(* Logix 5000 project; controller test_calc vendor 1 type 14 code 106 rev 31.11; software revision 31.01 *)

TASK MainTask (continuous, watchdog 500 ms) : MainProgram

MODULES
   Local : vendor 1 type 14 code 106 (Compact 0, rev 31.11)
END_MODULES

VAR_GLOBAL   (* controller tags *)
   cyc_h : REAL;
   cyl_h : REAL;
   cyl_rad : REAL;
   GAL : REAL;
END_VAR

PROGRAM MainProgram   (* main routine MainRoutine *)

ROUTINE calc   (* structured text *)
   pi*cyl_rad^2-cyl_rad^2*ACOS((cyl_rad-cyl_h)/cyl_rad)+(cyl_rad-cyl_h)*SQRT(2*cyl_rad*cyl_h-cyl_h^2)==GAL
END_ROUTINE

ROUTINE MainRoutine   (* ladder *)
END_ROUTINE
END_PROGRAM
